{attribute 'qualified_only'}
{attribute 'strict'}
TYPE LogEventLevel :
(	
    Verbose := 0,
    Debug,
    Information,
    Warning,
    Error,
    Fatal
);
END_TYPE

(* stored: Version 1.1.0.1, ProductVersion 3.1.4024.3
   DUT LogEventLevel: Id {327e4579-1840-4632-8c93-afe30595720f} *)
